FUNCTION_BLOCK TcoInspectionGroupTests EXTENDS TcoCore._internals_TcoContext
VAR
    _sut                 : TcoInspectors.TcoInspectionGroup(THIS^, TcoCore.NO.Structure);
    _diis                : ARRAY[0..1] OF TcoInspectors.TcoDigitalInspector(THIS^, TcoCore.NO.Structure);
    _dii_inspectedValues : ARRAY[0..1] OF BOOL;
    _dais                : ARRAY[0..1] OF TcoInspectors.TcoAnalogueInspector(THIS^, TcoCore.NO.Structure);
    _dai_inspectedValues : ARRAY[0..1] OF REAL;
    _ddis                : ARRAY[0..1] OF TcoInspectors.TcoDataInspector(THIS^, TcoCore.NO.Structure);
    _ddi_inspectedValues : ARRAY[0..1] OF STRING;
    _overallResult       : TcoInspectors.TcoComprehensiveResult;
    _coordinator         : MockCoordinator;
    _retryState          : INT;
END_VAR

METHOD PROTECTED Main
CASE _testId OF
    eInspectionGroupTests.Inspect:
         THIS^.ProbeDoneWhen(_sut.Act(_overallResult)
                 .Inspect(_diis[0].Inspect(_dii_inspectedValues[0]))
                 .Inspect(_diis[1].Inspect(_dii_inspectedValues[1]))
                 .Inspect(_dais[0].Inspect(_dai_inspectedValues[0]))
                 .Inspect(_dais[1].Inspect(_dai_inspectedValues[1]))
                 .Inspect(_ddis[0].Inspect(_ddi_inspectedValues[0]))
                 .Inspect(_ddis[1].Inspect(_ddi_inspectedValues[1]))
                 .UpdateComprehensiveResult(_overallResult).Done);
    eInspectionGroupTests.OnFailCarryOn:
        THIS^.ProbeDoneWhen(_sut.Act(_overallResult)
                .Inspect(_diis[0].Inspect(_dii_inspectedValues[0]))
                .Inspect(_diis[1].Inspect(_dii_inspectedValues[1]))
                .Inspect(_dais[0].Inspect(_dai_inspectedValues[0]))
                .Inspect(_dais[1].Inspect(_dai_inspectedValues[1]))
                .Inspect(_ddis[0].Inspect(_ddi_inspectedValues[0]))
                .Inspect(_ddis[1].Inspect(_ddi_inspectedValues[1]))
                .UpdateComprehensiveResult(_overallResult)
                .OnFail(_coordinator)
                .CarryOn());
    eInspectionGroupTests.OnFailRetry:
        THIS^.ProbeDoneWhen(_sut.Act(_overallResult)
                .Inspect(_diis[0].Inspect(_dii_inspectedValues[0]))
                .Inspect(_diis[1].Inspect(_dii_inspectedValues[1]))
                .Inspect(_dais[0].Inspect(_dai_inspectedValues[0]))
                .Inspect(_dais[1].Inspect(_dai_inspectedValues[1]))
                .Inspect(_ddis[0].Inspect(_ddi_inspectedValues[0]))
                .Inspect(_ddis[1].Inspect(_ddi_inspectedValues[1]))
                .UpdateComprehensiveResult(_overallResult)
                .OnFail(_coordinator)
                .Retry(_retryState));
    eInspectionGroupTests.OnFailTerminate:
        THIS^.ProbeDoneWhen(_sut.Act(_overallResult)
                .Inspect(_diis[0].Inspect(_dii_inspectedValues[0]))
                .Inspect(_diis[1].Inspect(_dii_inspectedValues[1]))
                .Inspect(_dais[0].Inspect(_dai_inspectedValues[0]))
                .Inspect(_dais[1].Inspect(_dai_inspectedValues[1]))
                .Inspect(_ddis[0].Inspect(_ddi_inspectedValues[0]))
                .Inspect(_ddis[1].Inspect(_ddi_inspectedValues[1]))
                .UpdateComprehensiveResult(_overallResult)
                .OnFail(_coordinator)
                .Terminate());
END_CASE
END_METHOD

END_FUNCTION_BLOCK

(* stored: Version 1.1.0.1, ProductVersion 3.1.4024.9
   POU TcoInspectionGroupTests: Id {982692a5-9906-0157-21ab-dccd4c43da53}, SpecialFunc None
   Method Main: Id {50a6684e-9742-0c51-2cf7-ef891467b3d3} *)
